(* IEC 61131-3 sources: DirIOWrap/, 3 files *)

(* ---- DirIOWrap.typ ---- *)
(********************************************************************
 * COPYRIGHT --
 ********************************************************************
 * Library: DirIOWrap
 * File: DirIOWrap.typ
 * Author: Josh
 * Created: April 24, 2015
 ********************************************************************
 * Data types of library DirIOWrap
 ********************************************************************)

TYPE
	DIOWrap_Int_FUB_typ : 	STRUCT
		Create : DirCreate; (*Open a file and read its contents*)
		Rename : DirRename; (*Open a file and read its contents*)
		Copy : DirCopy; (*Open a file and read its contents*)
		Delete : DirDeleteEx; (*Open a file and read its contents*)
		RenameFile : FileRename; (*Open a file and read its contents*)
		CopyFile : FileCopy; (*Open a file and read its contents*)
		DeleteFile : FileDelete; (*Open a file and read its contents*)
		ConvertToFile : DataObjToFile;
		ConvertToDataObject : FileToDataObj;
		Zip : DIODelegate_typ;
		Unzip : DIODelegate_typ;
		ConvertFolderToDataObject : DIODelegate_typ;
		ConvertToFolder : DIODelegate_typ;
	END_STRUCT;
	DIOWrap_Internal_typ : 	STRUCT
		FUB : DIOWrap_Int_FUB_typ;
		CMD : DIOWrap_IN_CMD_typ;
		NewFileIndex : UDINT;
		SrcName : STRING[DIOWRAP_STRLEN_NAME];
		DstName : STRING[DIOWRAP_STRLEN_NAME];
	END_STRUCT;
	DIOWrap_OUT_STAT_typ : 	STRUCT
		Busy : BOOL;
		Done : BOOL;
		Error : BOOL;
		ErrorID : UINT;
		ErrorString : STRING[DIOWRAP_STRLEN_ERROR];
	END_STRUCT;
	DIOWrap_OUT_typ : 	STRUCT
		STAT : DIOWrap_OUT_STAT_typ;
	END_STRUCT;
	DIOWrap_IN_PAR_typ : 	STRUCT
		SrcDevice : STRING[DIOWRAP_STRLEN_NAME]; (*File device name*)
		SrcPath : STRING[DIOWRAP_STRLEN_NAME]; (*File name (with extension)*)
		SrcName : STRING[DIOWRAP_STRLEN_NAME]; (*File name (with extension)*)
		DestDevice : STRING[DIOWRAP_STRLEN_NAME]; (*File device name*)
		DestPath : STRING[DIOWRAP_STRLEN_NAME]; (*File name (with extension)*)
		DestName : STRING[DIOWRAP_STRLEN_NAME]; (*File name (with extension)*)
	END_STRUCT;
	DIOWrap_IN_CMD_typ : 	STRUCT
		CreateDirectory : BOOL; (*Open a file and read its contents*)
		Rename : BOOL; (*Open a file and read its contents*)
		Copy : BOOL; (*Open a file and read its contents*)
		Move : BOOL;
		Delete : BOOL; (*Open a file and read its contents*)
		ConvertToFile : BOOL; (*Open a file and read its contents*)
		ExtractDataObject : BOOL; (*Open a file and read its contents*)
		ConvertToDataObject : BOOL; (*Open a file and read its contents*)
		Zip : BOOL; (*Open a file and read its contents*)
		Unzip : BOOL; (*Open a file and read its contents*)
	END_STRUCT;
	DIOWrap_IN_typ : 	STRUCT
		CMD : DIOWrap_IN_CMD_typ;
		PAR : DIOWrap_IN_PAR_typ;
	END_STRUCT;
	DIOWrap_typ : 	STRUCT
		IN : DIOWrap_IN_typ;
		OUT : DIOWrap_OUT_typ;
		Internal : DIOWrap_Internal_typ;
	END_STRUCT;
	DIODelegate_typ : 	STRUCT
		Active : BOOL;
		enable : BOOL;
		Execute : USINT;
		DataObjectName : STRING[10];
		FileDevice : STRING[20];
		FileName : STRING[80];
		TempFileDevice : STRING[20];
		Status : UINT;
		DestPath : STRING[80];
	END_STRUCT;
	LoadFileVolatile_internal_typ : 	STRUCT
		FileOpen : FileOpen;
		FileRead : FileRead;
		FileClose : FileClose;
		AllocStatus : UINT;
		_Open : BOOL;
		_Active : BOOL;
	END_STRUCT;
	LoadDatObjVolatile_internal_typ : 	STRUCT
		DatObjInfo : DatObjInfo;
		DatObjRead : DatObjRead;
		AllocStatus : UINT;
		_Active : BOOL;
	END_STRUCT;
	DeleteDatObj_internal_typ : 	STRUCT
		DatObjInfo : DatObjInfo;
		DatObjDelete : DatObjDelete;
		_Active : BOOL;
		_Execute : BOOL;
	END_STRUCT;
	DataObjToFile_internal_typ : 	STRUCT
		ReadDataObject : ReadDataObjectVolatile;
		CreateFile : CreateFile;
		_Execute : BOOL;
	END_STRUCT;
	FileToDataObj_internal_typ : 	STRUCT
		ReadFile : ReadFileVolatile;
		CreateDataObject : CreateDataObject;
		DataLength : UDINT;
		AllocStatus : UINT;
		pData : UDINT;
		_Execute : BOOL;
		_Active : BOOL;
	END_STRUCT;
	CreateWriteFile_internal_typ : 	STRUCT
		FileCreate : FileCreate;
		FileWrite : FileWrite;
		FileClose : FileClose;
		_Active : BOOL;
		_Open : BOOL;
		_Execute : BOOL;
	END_STRUCT;
	CreateDataObject_internal_typ : 	STRUCT
		CreateDataObject : DatObjCreate;
		_Execute : BOOL;
	END_STRUCT;
	AppendDataObject_internal_typ : 	STRUCT
		ReadDataObject : ReadDataObjectVolatile;
		DeleteDataObject : DeleteDataObject;
		WriteDataObject : CreateDataObject;
		DataLength : UDINT;
		pData : UDINT;
		AllocStatus : UINT;
		_Execute : BOOL;
		_Active : BOOL;
	END_STRUCT;
	DataObjectFileHeader_typ : 	STRUCT
		HEAD : STRING[7] := 'File';
		FileName : STRING[80];
		FileSize : UDINT;
	END_STRUCT;
END_TYPE

(* ---- DirIOWrap.fun ---- *)
(********************************************************************
 * COPYRIGHT --
 ********************************************************************
 * Library: DirIOWrap
 * File: DirIOWrap.fun
 * Author: Josh
 * Created: April 24, 2015
 ********************************************************************
 * Functions and function blocks of library DirIOWrap
 ********************************************************************)

FUNCTION DirIO : UINT (*Wrapper for common directory functions*) (*$GROUP=User*)
	VAR_IN_OUT
		t : DIOWrap_typ;
	END_VAR
END_FUNCTION

FUNCTION ValidDirectoryName : BOOL (*TODO: Add your comment here*) (*$GROUP=User*)
	VAR_INPUT
		Name : UDINT;
	END_VAR
END_FUNCTION

FUNCTION_BLOCK ReadFileVolatile (*TODO: Add your comment here*) (*$GROUP=User*)
	VAR_INPUT
		Enable : BOOL;
		FileDevice : STRING[80];
		FileName : STRING[80];
	END_VAR
	VAR_OUTPUT
		pData : UDINT;
		DataLen : UDINT;
		Status : UINT;
	END_VAR
	VAR
		internal : LoadFileVolatile_internal_typ;
	END_VAR
END_FUNCTION_BLOCK

FUNCTION_BLOCK ReadDataObjectVolatile (*TODO: Add your comment here*) (*$GROUP=User*)
	VAR_INPUT
		Enable : BOOL;
		DataObjectName : STRING[10];
	END_VAR
	VAR_OUTPUT
		pData : UDINT;
		DataLen : UDINT;
		Status : UINT;
	END_VAR
	VAR
		internal : LoadDatObjVolatile_internal_typ;
	END_VAR
END_FUNCTION_BLOCK

FUNCTION_BLOCK DeleteDataObject (* *) (*$GROUP=User,$CAT=User,$GROUPICON=User.png,$CATICON=User.png*)
	VAR_INPUT
		Execute : BOOL;
		DataObjectName : STRING[10];
	END_VAR
	VAR_OUTPUT
		Status : UINT;
	END_VAR
	VAR
		internal : DeleteDatObj_internal_typ;
	END_VAR
END_FUNCTION_BLOCK

FUNCTION_BLOCK CreateFile (*Create a file and write data to it*) (*$GROUP=User,$CAT=User,$GROUPICON=User.png,$CATICON=User.png*)
	VAR_INPUT
		Execute : BOOL;
		FileDevice : STRING[80];
		FileName : STRING[80];
		pData : UDINT;
		DataLen : UDINT;
	END_VAR
	VAR_OUTPUT
		Status : UINT;
	END_VAR
	VAR
		internal : CreateWriteFile_internal_typ;
	END_VAR
END_FUNCTION_BLOCK

FUNCTION_BLOCK FileToDataObj (*Convert dataobject to file*) (*$GROUP=User,$CAT=User,$GROUPICON=User.png,$CATICON=User.png*)
	VAR_INPUT
		Execute : BOOL;
		FileDevice : STRING[80];
		FileName : STRING[80];
		DataObjectName : STRING[10];
	END_VAR
	VAR_OUTPUT
		Status : UINT;
	END_VAR
	VAR
		internal : FileToDataObj_internal_typ;
	END_VAR
END_FUNCTION_BLOCK

FUNCTION_BLOCK DataObjToFile (*Convert a file to a dataobject*) (*$GROUP=User,$CAT=User,$GROUPICON=User.png,$CATICON=User.png*)
	VAR_INPUT
		Execute : BOOL;
		FileDevice : STRING[80];
		FileName : STRING[80];
		DataObjectName : STRING[10];
	END_VAR
	VAR_OUTPUT
		ExportFileName : STRING[80];
		Status : UINT;
	END_VAR
	VAR
		internal : DataObjToFile_internal_typ;
	END_VAR
END_FUNCTION_BLOCK

FUNCTION_BLOCK CreateDataObject (*Create Data object from data*) (*$GROUP=User,$CAT=User,$GROUPICON=User.png,$CATICON=User.png*)
	VAR_INPUT
		Execute : BOOL;
		DataObjectName : STRING[10];
		pData : UDINT;
		DataLen : UDINT;
	END_VAR
	VAR_OUTPUT
		Status : UINT;
	END_VAR
	VAR
		internal : CreateDataObject_internal_typ;
	END_VAR
END_FUNCTION_BLOCK

FUNCTION_BLOCK AppendDataObject (* *) (*$GROUP=User,$CAT=User,$GROUPICON=User.png,$CATICON=User.png*)
	VAR_INPUT
		Execute : BOOL;
		DataObjectName : STRING[10];
		pData : UDINT;
		DataLen : UDINT;
	END_VAR
	VAR_OUTPUT
		Status : UINT;
	END_VAR
	VAR
		internal : AppendDataObject_internal_typ;
	END_VAR
END_FUNCTION_BLOCK

(* ---- DirIOWrap.var ---- *)
(********************************************************************
 * COPYRIGHT --
 ********************************************************************
 * Library: DirIOWrap
 * File: DirIOWrap.var
 * Author: Josh
 * Created: April 24, 2015
 ********************************************************************
 * Constants of library DirIOWrap
 ********************************************************************)
VAR CONSTANT
	DIOWRAP_STRLEN_ERROR : USINT := 80;
	DIOWRAP_STRLEN_NAME : UINT := 260;
	DIOWRAP_STAT_OK : UINT := 0;
	DIOWRAP_STAT_DISABLED : UINT := 65534;
END_VAR
